PROGRAM pouS1Alarms
VAR
	

END_VAR

// NETWORK 1

END_PROGRAM

(* stored: Version 1.1.0.1, ProductVersion 3.1.4024.12
   POU pouS1Alarms: Id {4e168d6b-ccd5-440b-8127-bea095611032}, SpecialFunc None *)
